{attribute 'pack_mode' := '1'} 
TYPE ST_TxRxMessage :
STRUCT
	dataLength : UINT;
	cobId : UDINT;
	data : ARRAY[0..7] OF BYTE;
END_STRUCT
END_TYPE

(* stored: Version 1.1.0.1, ProductVersion 3.1.4024.9
   DUT ST_TxRxMessage: Id {dead949c-ab50-4d2e-b6e4-d3f0529dda37} *)
